// TwinCAT 3 PLC project Readme
// ProgramVersion: 3.1.4023.0
// libraries:
//   Tc2_Standard, * (Beckhoff Automation GmbH)
//   Tc2_System, * (Beckhoff Automation GmbH)
//   Tc3_Module, * (Beckhoff Automation GmbH)
//   TcoCognexVision, * (Vortex.Library)
//   TcoCore, * (Vortex.Library)
// project tree:
//   GVLs/ GVL.TcGVL
//   / PlcTask.TcTTO
//   POUs/ MAIN.TcPOU, myVeryFirstTcoContext.TcPOU

CONFIGURATION Readme
    RESOURCE PLC ON TwinCAT3
        TASK PlcTask(INTERVAL := T#10ms, PRIORITY := 22);
        PROGRAM MAIN WITH PlcTask : MAIN;
    END_RESOURCE
END_CONFIGURATION

// ---- GVLs/GVL.TcGVL
{attribute 'qualified_only'}
VAR_GLOBAL
    myVeryFirstDatamanGVL : TcoCognexVision.TcoDatamanIO_v_5_x_x;
END_VAR

// ---- POUs/MAIN.TcPOU
PROGRAM MAIN
VAR
END_VAR

myVeryFirstTcoContext.Run();

END_PROGRAM

// ---- POUs/myVeryFirstTcoContext.TcPOU
FUNCTION_BLOCK myVeryFirstTcoContext EXTENDS TcoCore.TcoContext
VAR
    {attribute addProperty Name "<#Enter user friendly name of this instance here!!!#>"}
    myVeryFirstDataman : TcoCognexVision.TcoDataman_v_5_x_x(THIS^);
END_VAR

(*~
    <docu>
        <summary>
            Main method of the TcoContext. This is the entry point of any control logic that belongs to this context.
            The call of this method is ensured by calling the <c>InstanceName.Run()</c> method, and it must not be called explicitly.
            This method is abstract, and it must be overridden in derived block.
        </summary>
    </docu>
~*)
METHOD PROTECTED Main
myVeryFirstDataman(inoIoData := GVL.myVeryFirstDatamanGVL);
myVeryFirstDataman.Service();
END_METHOD

END_FUNCTION_BLOCK
